# B&R Automation Studio project soft_bellows_measurement
Automation Studio 4.9

## Configuration Config1

CPU 4PPC70.0702-20B, AutomationRuntime B4.93, Build 4.1.2, Vc V4.72.6

### Task classes (Cpu.sw)
```
Cyclic#1:
  Measuremen <- Source.Measurement.prg
VcDataObjects: Visu <- Visu.dob
Binaries: vcpfppc7, vccalarm, vcnet, udbdef, vcrt, vcpkat, vccbar, vccurl, vcchtml, vccslider, Visu03, vcfile, vcpdihd, vcgclass, vccstr, vcpdsw, arial, vccbmp, vcmgr, vcshared, vcpdi855, vcctrend, vcchspot, vcdsloc, vcctext, Visu02, vcpdi815, vccovl, vcfntttf, arialbd, vcalarm, vcptelo, vccdt, vccline, vccbtn, vcpdvnc, vcbclass, vcxml, vcdsint, vctcal, TCData, FWRules, vcpk, vccnum, Visu01, iomap, asfw, Role, ashwac, sysconf, ashwd, User, arconfig
Libraries: standard, runtime, sys_lib, vcresman, asieccon, fileio, astime, dataobj
```

### Hardware
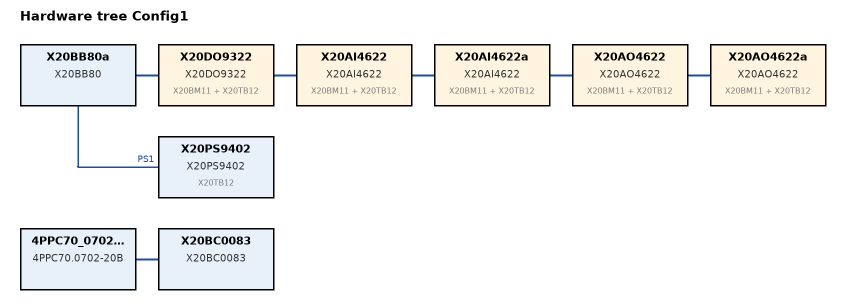
```
4PPC70_0702_20B : 4PPC70.0702-20B v1.6.1.0
  Connector IF2:
    ActivateDevice = 1
    Mode = Manual
    InternetAddress = 192.168.1.100
    SubnetMask = 255.255.255.0
    Vnc1
    VncVcObjectName1 = Visu
    VncKeyMappingFile1 = VC\PS2-Keyboard.dis
  ConfigurationID = icra2024_measurements_Config1
  FileDevice1
  FileDeviceName1 = USER
  FileDevicePath1 = USER_PATH
  VcObjectName = Visu
  KeyMappingFile = VC\4PPC70_0702_20B.dis
X20AI4622 : X20AI4622 v1.2.0.0  [SS1 -> X20TB12c.SS; SL -> X20BM11b.SL1]
X20AI4622a : X20AI4622 v1.2.0.0  [SS1 -> X20TB12d.SS; SL -> X20BM11c.SL1]
X20AO4622 : X20AO4622 v1.3.0.0  [SS1 -> X20TB12e.SS; SL -> X20BM11d.SL1]
X20AO4622a : X20AO4622 v1.3.0.0  [SS1 -> X20TB12f.SS; SL -> X20BM11e.SL1]
X20BB80a : X20BB80 v1.1.0.0
X20BC0083 : X20BC0083 v2.14.0.0  [PLK1 -> 4PPC70_0702_20B.IF1 (NodeNumber=1) [Cable Type=PowerlinkCable, Length=10, Version=1.0.0.3]; SL -> X20BB80a.SL1]
X20BM11a : X20BM11 v1.1.0.0  [X2X1 -> X20BB80a.IF1]
X20BM11b : X20BM11 v1.1.0.0  [X2X1 -> X20BM11a.X2X2]
X20BM11c : X20BM11 v1.1.0.0  [X2X1 -> X20BM11b.X2X2]
X20BM11d : X20BM11 v1.1.0.0  [X2X1 -> X20BM11c.X2X2]
X20BM11e : X20BM11 v1.1.0.0  [X2X1 -> X20BM11d.X2X2]
X20DO9322 : X20DO9322 v1.5.0.0  [SS1 -> X20TB12a.SS; SL -> X20BM11a.SL1]
X20PS9402 : X20PS9402 v1.2.0.0  [SS1 -> X20TB12b.SS; PS -> X20BB80a.PS1]
X20TB12a : X20TB12 v1.0.0.0
X20TB12b : X20TB12 v1.0.0.0
X20TB12c : X20TB12 v1.0.0.0
X20TB12d : X20TB12 v1.0.0.0
X20TB12e : X20TB12 v1.0.0.0
X20TB12f : X20TB12 v1.0.0.0
```

### IoMap.iom - 4PPC70_0702_20B/IoMap.iom
```iecst
VAR_CONFIG
	::valve.valve[0] AT %QW."X20AO4622".AnalogOutput01;
	::valve.valve[1] AT %QW."X20AO4622".AnalogOutput02;
	::valve.valve[2] AT %QW."X20AO4622".AnalogOutput03;
	::valve.valve[3] AT %QW."X20AO4622".AnalogOutput04;
	::sensor.bellow[0] AT %IW."X20AI4622a".AnalogInput01;
	::sensor.bellow[1] AT %IW."X20AI4622a".AnalogInput02;
	::sensor.bellow[2] AT %IW."X20AI4622a".AnalogInput03;
	::sensor.bellow[3] AT %IW."X20AI4622a".AnalogInput04;
END_VAR
```

## Logical view

### Global.typ
```iecst
TYPE
	valves : 	STRUCT
		valve : ARRAY[0..3]OF INT;
	END_STRUCT;
	sensors : 	STRUCT
		bellow : ARRAY[0..3]OF INT;
		voltage : ARRAY[0..3]OF REAL;
	END_STRUCT;
	measurement_parameters : 	STRUCT
		number_of_cycles : INT;
		time : INT := 1500;
		start : BOOL;
		timer_start : BOOL;
		step : INT := 0;
		desired_pressures : ARRAY[0..3]OF REAL := [3,4,5,6];
		done : INT;
		pressures : ARRAY[0..3]OF REAL;
		actual_cycle : INT := 1;
		remaining_time : INT;
	END_STRUCT;
END_TYPE
```

### Global.var
```iecst
VAR
	measurement : measurement_parameters;
	sensor : sensors;
	valve : valves;
END_VAR
```

### Program Logical/Source/Measurement (IEC)

#### Variables.var
```iecst
VAR
	TON_0 : TON;
	i : INT;
	a : UINT;
END_VAR
```

#### Cyclic.st
```iecst
PROGRAM _CYCLIC

	TON_0(IN := measurement.timer_start, PT := INT_TO_TIME(measurement.time));

	CASE measurement.step OF

		0:
			// Waiting for Start button press
			IF measurement.start = TRUE THEN
				measurement.actual_cycle	:= 1;
				FOR i:=0 TO 3 BY 1 DO
					valve.valve[i]			:= 0;			// zero pressure to all valves
				END_FOR
				measurement.step			:= 1;
			END_IF

		1:
			IF measurement.start = FALSE THEN
				FOR i:=0 TO 3 BY 1 DO
					valve.valve[i]		:= 0;			// zero pressure to all valves
				END_FOR
			ELSE
				// Set pressure for all valves
				measurement.timer_start	:= TRUE;		// start timer
				FOR i:=0 TO 3 BY 1 DO
					measurement.pressures[i]:= measurement.desired_pressures[i]*32767/9;
					valve.valve[i]			:= REAL_TO_INT(measurement.pressures[i]);
				END_FOR
				measurement.step			:= 2;			// next step
			END_IF

		2:
			// Waiting for timer
			IF TON_0.Q = TRUE THEN
				measurement.timer_start	:= FALSE;
				FOR i:=0 TO 3 BY 1 DO
					sensor.voltage[i]	:= INT_TO_REAL(sensor.bellow[i])*10/32767;
				END_FOR
				measurement.done		:= 1;
				measurement.step		:= 3;
			END_IF

		3:
			// Zero valves pressure
			measurement.done			:= 0;
			FOR i:=0 TO 3 BY 1 DO
				valve.valve[i]			:= 0;
			END_FOR
			measurement.step			:= 4;
			measurement.timer_start		:= TRUE;

		4:

			//Waiting for timer
			IF TON_0.Q = TRUE THEN
				measurement.timer_start	:= FALSE;
				measurement.step		:= 1;
				measurement.actual_cycle:= measurement.actual_cycle + 1;
				IF measurement.actual_cycle > measurement.number_of_cycles THEN
					measurement.start		:= FALSE;
					measurement.step		:= 5;
				END_IF
			END_IF

		5:
			IF measurement.start = FALSE THEN
				measurement.step			:= 0;
			END_IF

	END_CASE

END_PROGRAM
```
